{attribute 'qualified_only'}
{attribute 'strict'}
TYPE E_PowerAction :
(
	NONE, 
	SHUTDOWN, 
	REBOOT
);
END_TYPE

(* stored: Version 1.1.0.1, ProductVersion 3.1.4024.15
   DUT E_PowerAction: Id {e6b09f51-df7c-4436-9a24-1b635a0bd834} *)
